(* PLC project Beremiz non-standard POUs library, Beremiz Beremiz 0.0 *)
(* stored: creationDateTime 2008-12-14T16:53:26, modificationDateTime 2014-03-17T08:07:24 *)

FUNCTION_BLOCK python_eval
  VAR_INPUT
    TRIG : BOOL;
    CODE : STRING;
  END_VAR
  VAR_OUTPUT
    ACK : BOOL;
    RESULT : STRING;
  END_VAR
  VAR
    STATE : DWORD;
    BUFFER : STRING;
    PREBUFFER : STRING;
    TRIGM1 : BOOL;
    TRIGGED : BOOL;
  END_VAR

            {extern void __PythonEvalFB(int, PYTHON_EVAL*);__PythonEvalFB(0, data__);}
          
END_FUNCTION_BLOCK

FUNCTION_BLOCK python_poll
  VAR_INPUT
    TRIG : BOOL;
    CODE : STRING;
  END_VAR
  VAR_OUTPUT
    ACK : BOOL;
    RESULT : STRING;
  END_VAR
  VAR
    STATE : DWORD;
    BUFFER : STRING;
    PREBUFFER : STRING;
    TRIGM1 : BOOL;
    TRIGGED : BOOL;
  END_VAR

            {extern void __PythonEvalFB(int, PYTHON_EVAL*);__PythonEvalFB(1,(PYTHON_EVAL*)(void*)data__);}
          
END_FUNCTION_BLOCK

FUNCTION_BLOCK python_gear
  VAR_INPUT
    N : UINT;
    TRIG : BOOL;
    CODE : STRING;
  END_VAR
  VAR_OUTPUT
    ACK : BOOL;
    RESULT : STRING;
  END_VAR
  VAR
    py_eval : python_eval;
    COUNTER : UINT;
  END_VAR
  VAR  (* added by the conversion: wires and edge detectors of the diagram *)
    _ADD10_OUT : UINT;
    _EQ13_OUT : BOOL;
  END_VAR

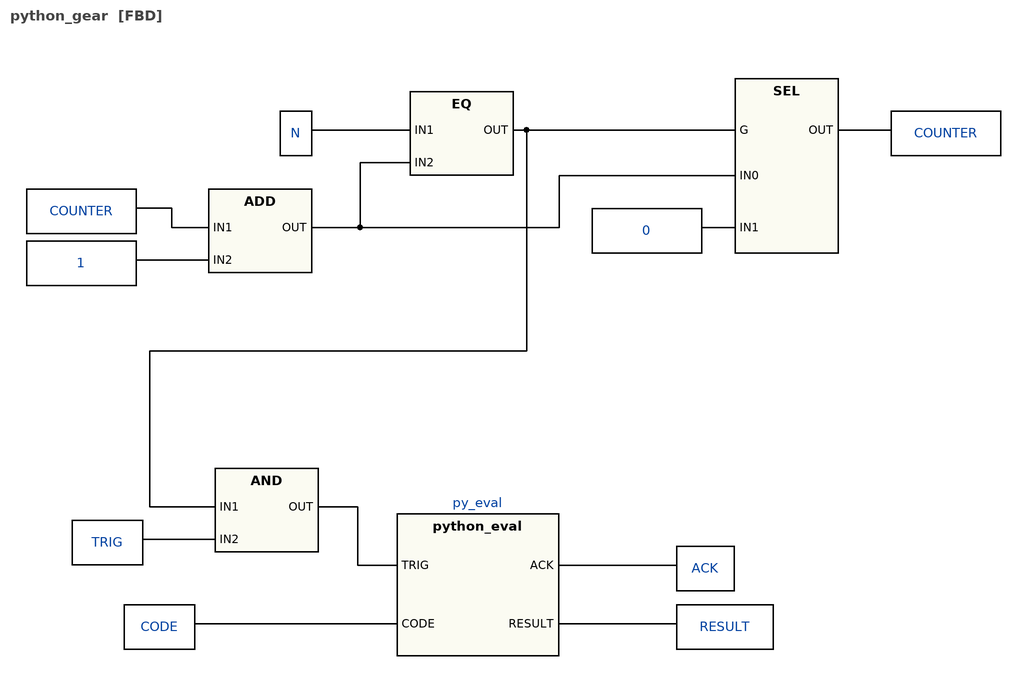
(* FBD diagram, written out as Structured Text *)
_ADD10_OUT := COUNTER + 1;
_EQ13_OUT := N = _ADD10_OUT;
COUNTER := SEL(_EQ13_OUT, _ADD10_OUT, 0);
py_eval(TRIG := _EQ13_OUT AND TRIG, CODE := CODE);
ACK := py_eval.ACK;
RESULT := py_eval.RESULT;
END_FUNCTION_BLOCK
